FUNCTION_BLOCK alarm
VAR_INPUT
	//Input that triggers the alarm condition
	trigger : BOOL;
	//Alarm Acknowledge bit, Clears low priority alarms
	alm_ack : BOOL;
	//Alarm Reset, clears high priority alarms
	reset : BOOL;
	//Alarm Priority, 1=Warning, 2=Error, 3=Critical
	priority : INT;
	//Alarm Delay Setpoint in Seconds
	delay_setpoint : REAL;
	//Alarm Enable
	enable : BOOL;
END_VAR
VAR_OUTPUT
	//Alarm is triggered
	active : BOOL;
	delay_ton_et : TIME;
END_VAR
VAR
	//Delay Timer Tags
	delay_ton : TON;
	delay_ton_pt : TIME;
	//delay_ton_et : TIME;
	//Delay setpoint converted to Milliseconds
	delay_ms : REAL;
	//Cutoff for needing to reset vs ack an alarm.  At or above this value requires reset.  
	reset_priority : REAL :=3;
END_VAR

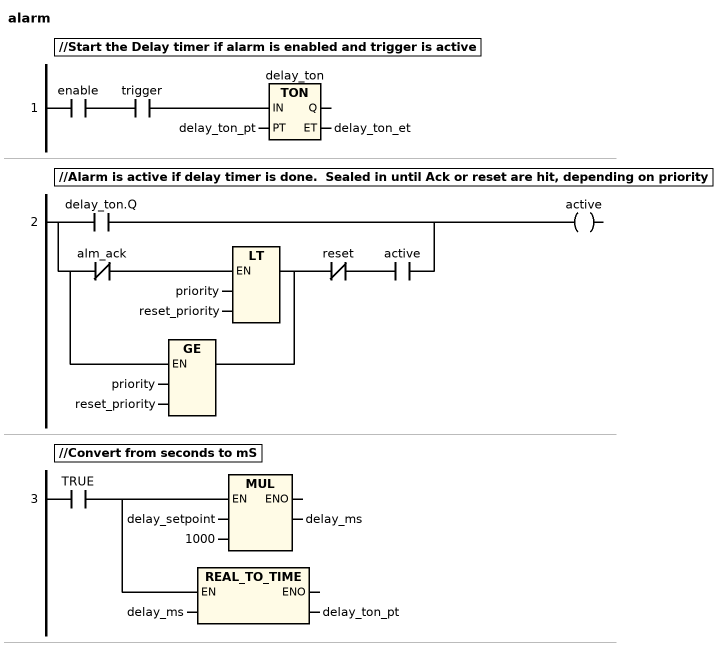
// NETWORK 1
// label: //Start the Delay timer if alarm is enabled and trigger is active
delay_ton(IN := enable AND trigger, PT := delay_ton_pt, ET => delay_ton_et); // TON

// NETWORK 2
// label: //Alarm is active if delay timer is done.  Sealed in until Ack or reset are hit, depending on priority
active := delay_ton.Q OR (NOT alm_ack AND priority < reset_priority OR priority >= reset_priority) AND NOT reset AND active;

// NETWORK 3
// label: //Convert from seconds to mS
delay_ms := delay_setpoint * 1000;
delay_ton_pt := REAL_TO_TIME(delay_ms);

END_FUNCTION_BLOCK

(* stored: Version 1.1.0.1, ProductVersion 3.1.4024.12
   POU alarm: Id {4941c71f-2070-4068-8b1d-744b33ae24df}, SpecialFunc None *)
